% RSLogix 500 project RTORES-200809-135922.RSS, saved by version 9.00.00.04 %
PROJECT "UNTITLED"    % processor: Bul.1763 MicroLogix 1100 Series B %

PROGRAM FILES
  LAD 2   4 rungs

DATA FILES
  O0 OUTPUT  4 elements
  I1 INPUT  6 elements
  S2 STATUS  66 elements
  B3 BINARY  1 elements
  T4 TIMER  2 elements
  C5 COUNTER  1 elements
  R6 CONTROL  1 elements
  N7 INTEGER  3 elements
  F8 FLOAT  1 elements
  ST9 STRINGS  4 elements

LADDER 2
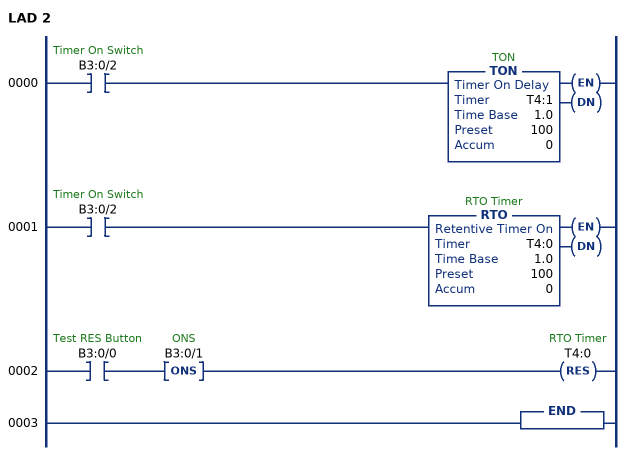
% Rung: 0 %
SOR XIC B3:0/2 TON T4:1 1.0 100 0 EOR
%   B3:0/2  "Timer On Switch" %
%   T4:1  "TON" %
% Rung: 1 %
SOR XIC B3:0/2 RTO T4:0 1.0 100 0 EOR
%   B3:0/2  "Timer On Switch" %
%   T4:0  "RTO Timer" %
% Rung: 2 %
SOR XIC B3:0/0 ONS B3:0/1 RES T4:0 EOR
%   B3:0/0  "Test RES Button" %
%   B3:0/1  "ONS" %
%   T4:0  "RTO Timer" %
% Rung: 3 %
SOR END EOR

OTHER DOCUMENTED ADDRESSES
  B3:0/3  "Test ABS Button"
  B3:0/4  "ONS"
  B3:0/5  "Test ASR Trigger Bit"
  N7:0  "0 = FALSE 1 = TRUE"
  N7:1  "Result Store"
  ST9:0  "Partial String 1"
  ST9:1  "Partial String 2"
  ST9:2  "Concatenated String"
  ST9:3  "Test Value"

DATA TABLE (non-zero values as saved)
DATA T4
% .PRE .ACC %
% T4:0 % 100 0
% T4:1 % 100 0
DATA ST9
% ST9:0 % "TEST"
% ST9:1 % "STRING"
% ST9:2 % "SOMETHING"
% ST9:3 % "TESTSTRING"
